  //============================= TRAN HEADER ==============================//
  // AUTOCODE   AUTOCODE   AUTOCODE   AUTOCODE   AUTOCODE   AUTOCODE   AUTO //
  // Bypass transition if manual jump:                                      //
  //------------------------------------------------------------------------//
      A #sqSequencer.STEP.Finished;
      A #smc.TRN_AND_JUMP   ;//Manual jump is set Transition as bypassed
      JCN COMM            ;//exit

NETWORK
TITLE = S016::STEP 016:TRAN 021: Empty Transition
//----------------------------------------------------------------------------//
// TRAN   TRAN   TRAN   TRAN   TRAN   TRAN   TRAN   TRAN   TRAN   TRAN   TRAN //
// TRAN   TRAN   TRAN   TRAN   TRAN   TRAN   TRAN   TRAN   TRAN   TRAN   TRAN //
//----------------------------------------------------------------------------//
// Empty Transition
//----------------------------------------------------------------------------//
// CONDITION   CONDITION   CONDITION   CONDITION   CONDITION   CONDITION   CO //
// CONDITION   CONDITION   CONDITION   CONDITION   CONDITION   CONDITION   CO //
//----------------------------------------------------------------------------//
      A "uncondJump";






  //============================= TRAN FOOTER ==============================//
  // Transition jump control:                                               //
  //------------------------------------------------------------------------//
      A #sqSequencer.STEP.JumpCtrl;
      S #sqSequencer.STEP.Jump;
      S #sqSequencer.STEP.jumpDone[16];

NETWORK
TITLE = S016:t021::TRANS-v: EXIT TRANSITION AND READY THE NEXT STEP
//------------------------------------------------------------------------//
// Check the jump flag and jump to the next step if the transition        //
// condition is true and has set the jump flag:                           //
//------------------------------------------------------------------------//
      A #sqSequencer.STEP.Jump;
      JCN x021;

      R #sqSequencer.STEP.Jump;
      R #sqSequencer.STEP.Finished;

      L 06   ;// Load next STEPNO to jump to if transition satisfied
      T #sqSequencer.STEP.NumberNext;//Next Step06.

      JU COMM            ;// Transition satisfied, Exit, go to next step
x021:      NOP 0;






NETWORK
TITLE = S016::STEP-016:EXIT TRANSITION:
//========================== STEP TRANSFER ===============================//
// Jump to the common step progression code:                              //
//------------------------------------------------------------------------//
      JU COMM;






NETWORK
TITLE = S017: STEP-17::UO_MX_SETUP : Break vacuum
//================================ STEP HEADER ===========================//
// STEP017 STEP017 STEP017 STEP017
// AUTOCODE   AUTOCODE   AUTOCODE   AUTOCODE   AUTOCODE   AUTOCODE   AUTO //
// STEP017 STEP017 STEP017 STEP017
//------------------------------------------------------------------------//
// Open HPCA supply valve to break the vacuum.
//------------------------------------------------------------------------//
S017:      NOP 0;

      SET;
      R #sqSequencer.STEP.jumpDone[17];
      A #sqSequencer.CMD.Pause;//If paused jump
      JC COMM;

NETWORK
TITLE = S017:STEP-17:Begin Action

      A #sqSequencer.STEP.Finished;
      JC A017;// Exit Action code, Jump to A017 Transition code

    //----------------------------------------------------------------------//
    // Begin step Action:                                                   //
    //----------------------------------------------------------------------//
      A #sqSequencer.STEP.Active;
      JC L017;// Action number loaded, Jump to L017--Step Action List

    //----------------------------------------------------------------------//
    // Load Default/Initial Step action number:                             //
    //----------------------------------------------------------------------//
      S #sqSequencer.STEP.Active;
      S #sqStepTimer.IN;
      L 1;//First Action, Step must contain Minimum one action
      T #sqSequencer.STEP.ActionNumber;

//----------------------------------------------------------------------------//
// Step action list.                                                          //
// aann=mini Action step number(aa) inside main step number(nn)               //
// First Action aa00, Second action ab00, Third ac00, etc.                    //
//----------------------------------------------------------------------------//
L017:      NOP 0;

      L #sqSequencer.STEP.ActionNumber;
      JL r017;//Wrong Action number
      JU _017;//Action error handling
      JU aa17;//ACTION-01
      JU ab17;//ACTION-02


//----------------------------------------------------------------------------//
// More step action in the list can be inserted here, upto ab is tested:      //
//----------------------------------------------------------------------------//
r017:      NOP 0;//Wrong action number
      S #sqSequencer.Error_Fault;
      JU k017;//Exit
_017:      NOP 0;// Action error handling
      JU k017;// Exit






NETWORK
TITLE = S017:: STEP-017:: : ACTION CODE
//================================ ACT HEADER ============================//
// ACTION ACTION ACTION ACTION ACTION ACTION ACTION ACTION ACTION ACTION  //
// AUTOCODE   AUTOCODE   AUTOCODE   AUTOCODE   AUTOCODE   AUTOCODE   AUTO //
// ACTION ACTION ACTION ACTION ACTION ACTION ACTION ACTION ACTION ACTION  //
//------------------------------------------------------------------------//
// //Open HPCA valve to break the vacuum
aa17:      NOP 0;

  //------------------------------------------------------------------------//
  // ACT ACT ACT ACT ACT ACT ACT ACT ACT ACT ACT ACT ACT ACT ACT ACT ACT    //
  //------------------------------------------------------------------------//
      L "dbCONST".SEL.GAS.HPCA;
      T #_emc_gas_medium_gas;
      L "dbCONST".BLK.CMD.RESTART;
      T #_emc_gas_cmd;

  //------------------------------------------------------------------------//
  // VERIFY  VERIFY VERIFY VERIFY VERIFY VERIFY VERIFY VERIFY VERIFY VERIFY //
  //------------------------------------------------------------------------//
      A(;
      L #_emc_gas_state;
      L "dbCONST".BLK.STATE.STOPPED;
      >I;
      );
      A(;
      L #_emc_gas_state;
      L "dbCONST".BLK.STATE.INTERLOCKED;
      <I;
      );
      S #sqSequencer.STEP.ActionVerified;//Action verified

  //------------------------------------------------------------------------//
  // Action done:                                                           //
  //------------------------------------------------------------------------//
      O #sqSequencer.STEP.ActionVerified;
      O #smc.NO_VERIFIC     ;//No verification , bypass verification code
      S #sqSequencer.STEP.ActionFinished;






  //============================= ACT FOOTER ===============================//
  // AUTOCODE   AUTOCODE   AUTOCODE   AUTOCODE   AUTOCODE   AUTOCODE   AUTO //
  // Get Ready after action finished:                                       //
  //------------------------------------------------------------------------//
      A #sqSequencer.STEP.ActionFinished;
      JCN k017;

  //------------------------------------------------------------------------//
  // Reset Action finished flag, ready for next step action:                //
  //------------------------------------------------------------------------//
      R #sqSequencer.STEP.ActionVerified;
      R #sqSequencer.STEP.ActionFinished;

  //------------------------------------------------------------------------//
  // Load Next Step Action number:                                          //
  //------------------------------------------------------------------------//
      L 02;//Load next Action
      T #sqSequencer.STEP.ActionNumber;






NETWORK
TITLE = S017:: STEP-017:: : ACTION CODE
//================================ ACT HEADER ============================//
// ACTION ACTION ACTION ACTION ACTION ACTION ACTION ACTION ACTION ACTION  //
// AUTOCODE   AUTOCODE   AUTOCODE   AUTOCODE   AUTOCODE   AUTOCODE   AUTO //
// ACTION ACTION ACTION ACTION ACTION ACTION ACTION ACTION ACTION ACTION  //
//------------------------------------------------------------------------//
// //Clear gas EM restart command
ab17:      NOP 0;

  //------------------------------------------------------------------------//
  // ACT ACT ACT ACT ACT ACT ACT ACT ACT ACT ACT ACT ACT ACT ACT ACT ACT    //
  //------------------------------------------------------------------------//
      L "dbCONST".BLK.CMD.START;
      T #_emc_gas_cmd;

  //------------------------------------------------------------------------//
  // VERIFY  VERIFY VERIFY VERIFY VERIFY VERIFY VERIFY VERIFY VERIFY VERIFY //
  //------------------------------------------------------------------------//

      S #sqSequencer.STEP.ActionVerified;//Action verified

  //------------------------------------------------------------------------//
  // Action done:                                                           //
  //------------------------------------------------------------------------//
      O #sqSequencer.STEP.ActionVerified;
      O #smc.NO_VERIFIC     ;//No verification , bypass verification code
      S #sqSequencer.STEP.ActionFinished;






  //============================= STEP FOOTER ==============================//
  // AUTOCODE   AUTOCODE   AUTOCODE   AUTOCODE   AUTOCODE   AUTOCODE   AUTO //
  // Get Ready after action finished:                                       //
  //------------------------------------------------------------------------//
      A #sqSequencer.STEP.ActionFinished;
      JCN k017;

  //------------------------------------------------------------------------//
  // Reset Action finished flag, ready for next step action:                //
  //------------------------------------------------------------------------//
      R #sqSequencer.STEP.ActionVerified;
      R #sqSequencer.STEP.ActionFinished;

  //------------------------------------------------------------------------//
  // If ALL actions are finished:                                           //
  //------------------------------------------------------------------------//
      SET;
      S #sqSequencer.STEP.Finished;
      R #sqSequencer.STEP.Active;
      S #sqSequencer.STEP.Done[17];

  //------------------------------------------------------------------------//
  // End Step action(s):                                                    //
  //------------------------------------------------------------------------//
      JU k017;

//----------------------------------------------------------------------------//
// Finished Step Action(s):                                                   //
//----------------------------------------------------------------------------//
k017:      NOP 0;

      A #sqStepTimerExpired;
      S #sqSequencer.STEP.WithError[17];// Step error flag
      S #sqSequencer.Error_Fault;
      R #sqStepTimer.IN;

NETWORK
TITLE = S017:STEP-017::Begin Transition
//------------------------------------------------------------------------//
// Begin the transition code:                                             //
//------------------------------------------------------------------------//
A017:      NOP 0;
      R #sqStepTimer.IN;






  //============================= TRAN HEADER ==============================//
  // AUTOCODE   AUTOCODE   AUTOCODE   AUTOCODE   AUTOCODE   AUTOCODE   AUTO //
  // Bypass transition if manual jump:                                      //
  //------------------------------------------------------------------------//
      A #sqSequencer.STEP.Finished;
      A #smc.TRN_AND_JUMP   ;//Manual jump is set Transition as bypassed
      JCN COMM            ;//exit

NETWORK
TITLE = S017::STEP 017:TRAN 022: Pressure at zero
//----------------------------------------------------------------------------//
// TRAN   TRAN   TRAN   TRAN   TRAN   TRAN   TRAN   TRAN   TRAN   TRAN   TRAN //
// TRAN   TRAN   TRAN   TRAN   TRAN   TRAN   TRAN   TRAN   TRAN   TRAN   TRAN //
//----------------------------------------------------------------------------//
// Pressure increased to 0
//----------------------------------------------------------------------------//
// CONDITION   CONDITION   CONDITION   CONDITION   CONDITION   CONDITION   CO //
// CONDITION   CONDITION   CONDITION   CONDITION   CONDITION   CONDITION   CO //
//----------------------------------------------------------------------------//
      O(;
      L #_emc_gas_pi_vessel_pv;
      L 0.0;
      >R;
      );






  //============================= TRAN FOOTER ==============================//
  // Transition jump control:                                               //
  //------------------------------------------------------------------------//
      A #sqSequencer.STEP.JumpCtrl;
      S #sqSequencer.STEP.Jump;
      S #sqSequencer.STEP.jumpDone[17];

NETWORK
TITLE = S017:t022::TRANS-v: EXIT TRANSITION AND READY THE NEXT STEP
//------------------------------------------------------------------------//
// Check the jump flag and jump to the next step if the transition        //
// condition is true and has set the jump flag:                           //
//------------------------------------------------------------------------//
      A #sqSequencer.STEP.Jump;
      JCN x022;

      R #sqSequencer.STEP.Jump;
      R #sqSequencer.STEP.Finished;

      L 18   ;// Load next STEPNO to jump to if transition satisfied
      T #sqSequencer.STEP.NumberNext;//Next Step18.

      JU COMM            ;// Transition satisfied, Exit, go to next step
x022:      NOP 0;






NETWORK
TITLE = S017::STEP-017:EXIT TRANSITION:
//========================== STEP TRANSFER ===============================//
// Jump to the common step progression code:                              //
//------------------------------------------------------------------------//
      JU COMM;






NETWORK
TITLE = S018: STEP-18::UO_MX_SETUP : Setup Unit Operation Completed
//================================ STEP HEADER ===========================//
// STEP018 STEP018 STEP018 STEP018
// AUTOCODE   AUTOCODE   AUTOCODE   AUTOCODE   AUTOCODE   AUTOCODE   AUTO //
// STEP018 STEP018 STEP018 STEP018
//------------------------------------------------------------------------//
// Clear used flags.
// Log Mx SETUP operation end time.
//------------------------------------------------------------------------//
S018:      NOP 0;

      SET;
      R #sqSequencer.STEP.jumpDone[18];
      A #sqSequencer.CMD.Pause;//If paused jump
      JC COMM;

NETWORK
TITLE = S018:STEP-18:Begin Action

      A #sqSequencer.STEP.Finished;
      JC A018;// Exit Action code, Jump to A018 Transition code

    //----------------------------------------------------------------------//
    // Begin step Action:                                                   //
    //----------------------------------------------------------------------//
      A #sqSequencer.STEP.Active;
      JC L018;// Action number loaded, Jump to L018--Step Action List

    //----------------------------------------------------------------------//
    // Load Default/Initial Step action number:                             //
    //----------------------------------------------------------------------//
      S #sqSequencer.STEP.Active;
      S #sqStepTimer.IN;
      L 1;//First Action, Step must contain Minimum one action
      T #sqSequencer.STEP.ActionNumber;

//----------------------------------------------------------------------------//
// Step action list.                                                          //
// aann=mini Action step number(aa) inside main step number(nn)               //
// First Action aa00, Second action ab00, Third ac00, etc.                    //
//----------------------------------------------------------------------------//
L018:      NOP 0;

      L #sqSequencer.STEP.ActionNumber;
      JL r018;//Wrong Action number
      JU _018;//Action error handling
      JU aa18;//ACTION-01


//----------------------------------------------------------------------------//
// More step action in the list can be inserted here, upto ab is tested:      //
//----------------------------------------------------------------------------//
r018:      NOP 0;//Wrong action number
      S #sqSequencer.Error_Fault;
      JU k018;//Exit
_018:      NOP 0;// Action error handling
      JU k018;// Exit






NETWORK
TITLE = S018:: STEP-018:: : ACTION CODE
//================================ ACT HEADER ============================//
// ACTION ACTION ACTION ACTION ACTION ACTION ACTION ACTION ACTION ACTION  //
// AUTOCODE   AUTOCODE   AUTOCODE   AUTOCODE   AUTOCODE   AUTOCODE   AUTO //
// ACTION ACTION ACTION ACTION ACTION ACTION ACTION ACTION ACTION ACTION  //
//------------------------------------------------------------------------//
// //Clear used flags.
// //Log Mx SETUP operation end time.
aa18:      NOP 0;

  //------------------------------------------------------------------------//
  // ACT ACT ACT ACT ACT ACT ACT ACT ACT ACT ACT ACT ACT ACT ACT ACT ACT    //
  //------------------------------------------------------------------------//
  // Stop gas
      L "dbCONST".BLK.CMD.STOP;
      T #_emc_gas_cmd;

//Clear used flags
      SET;
      R #_prompt_connect_ok;
      R #_prompt_connect_ok_confirm_yes;

//Log SETUP operation end time.
      SET;
      S #_log_msg_setup_end;

  //------------------------------------------------------------------------//
  // VERIFY  VERIFY VERIFY VERIFY VERIFY VERIFY VERIFY VERIFY VERIFY VERIFY //
  //------------------------------------------------------------------------//
      A "uncondJump";
      S #sqSequencer.STEP.ActionVerified;//Action verified

  //------------------------------------------------------------------------//
  // Action done:                                                           //
  //------------------------------------------------------------------------//
      O #sqSequencer.STEP.ActionVerified;
      O #smc.NO_VERIFIC     ;//No verification , bypass verification code
      S #sqSequencer.STEP.ActionFinished;






  //============================= STEP FOOTER ==============================//
  // AUTOCODE   AUTOCODE   AUTOCODE   AUTOCODE   AUTOCODE   AUTOCODE   AUTO //
  // Get Ready after action finished:                                       //
  //------------------------------------------------------------------------//
      A #sqSequencer.STEP.ActionFinished;
      JCN k018;

  //------------------------------------------------------------------------//
  // Reset Action finished flag, ready for next step action:                //
  //------------------------------------------------------------------------//
      R #sqSequencer.STEP.ActionVerified;
      R #sqSequencer.STEP.ActionFinished;

  //------------------------------------------------------------------------//
  // If ALL actions are finished:                                           //
  //------------------------------------------------------------------------//
      SET;
      S #sqSequencer.STEP.Finished;
      R #sqSequencer.STEP.Active;
      S #sqSequencer.STEP.Done[18];

  //------------------------------------------------------------------------//
  // End Step action(s):                                                    //
  //------------------------------------------------------------------------//
      JU k018;

//----------------------------------------------------------------------------//
// Finished Step Action(s):                                                   //
//----------------------------------------------------------------------------//
k018:      NOP 0;

      A #sqStepTimerExpired;
      S #sqSequencer.STEP.WithError[18];// Step error flag
      S #sqSequencer.Error_Fault;
      R #sqStepTimer.IN;

NETWORK
TITLE = S018:STEP-018::Begin Transition
//------------------------------------------------------------------------//
// Begin the transition code:                                             //
//------------------------------------------------------------------------//
A018:      NOP 0;
      R #sqStepTimer.IN;






NETWORK
TITLE = S018::STEP-018:EXIT TRANSITION:
//========================== STEP TRANSFER ===============================//
// Jump to the common step progression code:                              //
//------------------------------------------------------------------------//
      JU COMM;






NETWORK
TITLE = Sequencer Common Code, Execute in Each Scan
//============================ SEQ FOOTER ================================//
// AUTOCODE   AUTOCODE   AUTOCODE   AUTOCODE   AUTOCODE   AUTOCODE   AUTO //
// Common code to execute each scan:                                      //
//------------------------------------------------------------------------//
COMM:      NOP 0;

NETWORK
TITLE = Retentive/Non Retentive Selectable Run timer
      CALL #sqRunTimer
      (  TIME_H                      := #sqRunTimer.TIME_H ,
         TIME_M                      := #sqRunTimer.TIME_M ,
         TIME_S                      := #sqRunTimer.TIME_S ,
         ENABLE                      := #sqRunTimer.ENABLE ,
         RESET                       := #sqRunTimer.RESET ,
         PAUSE                       := #sqRunTimer.PAUSE ,
         NON_RET                     := #sqRunTimer.NON_RET ,
         RMNG_H                      := #sqRunTimer.RMNG_H ,
         RMNG_M                      := #sqRunTimer.RMNG_M ,
         RMNG_S                      := #sqRunTimer.RMNG_S ,
         TIME_EXPIRED                := #sqRunTimer.TIME_EXPIRED ,
         TMR_RUNNG                   := #sqRunTimer.TMR_RUNNG
      );

NETWORK
TITLE = Sequencer Step Timer
      CALL #sqStepTimer
      {time_type := 'Time'}
      (  IN                          := #sqStepTimer.IN ,
         PT                          := "dbCONST".SEQ.STEP_TIME ,
         Q                           := #sqStepTimerExpired ,
         ET                          := #sqStepTimerElapsed
      );

NETWORK
TITLE = Sequencer Timer
      CALL #SQ_TIMER
      {time_type := 'Time'}
      (  IN                          := #sqSeqTimerStart ,
         PT                          := #SQ_TIMER.PT ,
         Q                           := #sqSeqTimerExpired ,
         ET                          := #sqSeqTimerElapsed
      );

      CALL #SQ_TIMER2
      {time_type := 'Time'}
      (  IN                          := #sqSeqTimerStart2 ,
         PT                          := #SQ_TIMER2.PT ,
         Q                           := #sqSeqTimerExpired2 ,
         ET                          := #sqSeqTimerElapsed2
      );

NETWORK
TITLE = Sequencer Timer
      CALL #SQ_TIMER3
      {time_type := 'Time'}
      (  IN                          := #sqSeqTimerStart3 ,
         PT                          := #SQ_TIMER3.PT ,
         Q                           := #sqSeqTimerExpired3 ,
         ET                          := #sqSeqTimerElapsed3
      );

NETWORK
TITLE = General Assignments

      L #sqSequencer.STEP.NumberNext;
      T #smc.NXT_STEP;
      T #sqSequencer.STEP.NumberCurrent;
      T #smc.CURSTEP;

      A #sqSequencer.STEP.Active;
      = #smc.S_ACTIVE;

      A #sqSequencer.Error_Fault;
      = #smc.ERR_FAULT;

NETWORK
TITLE = Stop command completion
      A #smc.OFF_IDLE;
      A #sqSequencer.STEP.Done[18];
      AN #sqSequencer.STEP.WithError[18];
      JCN NotStopCmd;
      R #smc.PAUSED;
      R #sqSequencer.STEP.Error_Fault;
      R #sqSequencer.Error_Fault;
      L "dbCONST".SEQ.STATE.OFF_IDLE;
      T #smc.SQ_STATE;
NotStopCmd:      NOP 0;

      A #smc.OFF_IDLE;
      AN #sqSequencer.STEP.Done[18];
      AN #sqSequencer.STEP.WithError[18];
      JCN _stopAction;
      R #sqSequencer.STEP.Finished;
      R #smc.PAUSED;
      R #sqSequencer.STEP.Error_Fault;
      R #sqSequencer.Error_Fault;
_stopAction:      NOP 0;

NETWORK
TITLE = Sequencer Finished

      AN #smc.OFF_IDLE;
      AN #smc.PAUSED;
      A #sqSequencer.STEP.Done[18];
      = #sqSequencer.Finished;
      = #smc.SQ_FINISHED;
      JCN fnsd;
      L "dbCONST".SEQ.STATE.COMPLETED;
      T #smc.SQ_STATE;
      R #smc.PAUSED;
      R #sqSequencer.STEP.Error_Fault;
      R #sqSequencer.Error_Fault;
fnsd:      NOP 0;

  //------------------------------------------------------------------------//
  // Reset Finished flag if SQ OFF for Last step to scan:                   //
  //------------------------------------------------------------------------//
      A #smc.ABORTED;
      AN #sqSequencer.STEP.Done[18];
      AN #sqSequencer.STEP.WithError[18];
      JCN _abrt_end;
      R #sqSequencer.STEP.Finished;
      R #smc.PAUSED;
      R #sqSequencer.STEP.Error_Fault;
      R #sqSequencer.Error_Fault;
      L "dbCONST".SEQ.STATE.ABORTED;
      T #smc.SQ_STATE;
_abrt_end:      NOP 0;

  //------------------------------------------------------------------------//
  // Visio Common Code Begin:                                               //
  //------------------------------------------------------------------------//


//----------------------------------------------------------------------------//
// End of Sequencer:                                                          //
//----------------------------------------------------------------------------//
END_FUNCTION_BLOCK

